// TIA Portal V18 export
DATA_BLOCK "previousValues"   // DB19
{ S7_Optimized_Access := 'TRUE' }
VERSION : 0.1
// stored: AutoNumber true, DBAccessibleFromOPCUA true, DBAccessibleFromWebserver true, InstanceOfName UDT_actualValues, InstanceOfType UDT, IsOnlyStoredInLoadMemory false, IsWriteProtectedInAS false
"UDT_actualValues"
   // VAR RETAIN
   //    target { ExternalVisible := 'False'; ExternalWritable := 'False'} : DInt;
   //    actual { ExternalVisible := 'False'; ExternalWritable := 'False'} : DInt;
   //    ok { ExternalVisible := 'False'; ExternalWritable := 'False'} : DInt;
   //    difference { ExternalVisible := 'False'; ExternalWritable := 'False'} : DInt;
   //    counterTactTime { ExternalVisible := 'False'; ExternalWritable := 'False'} : DInt;
   //    state { ExternalVisible := 'False'; ExternalWritable := 'False'} : DInt;
   // END_VAR
BEGIN
END_DATA_BLOCK
